FUNCTION IO_TO_ATT : ST_PMPS_Attenuator
VAR_INPUT
    IO : ST_PMPS_Attenuator_IO;
END_VAR
VAR
END_VAR

IO_TO_ATT.nAtt := IO.nAtt;
IO_TO_ATT.xAttOK := IO.xAttOK;

END_FUNCTION

(* stored: Version 1.1.0.1, ProductVersion 3.1.4022.18
   POU IO_TO_ATT: Id {3894235d-c53a-42f8-8be8-70feba0a504b}, SpecialFunc None *)
